// LS Electric XG5000 project: 8_22_1
// PLC LSPLC

PROGRAM NewProgram (task: 스캔 프로그램)

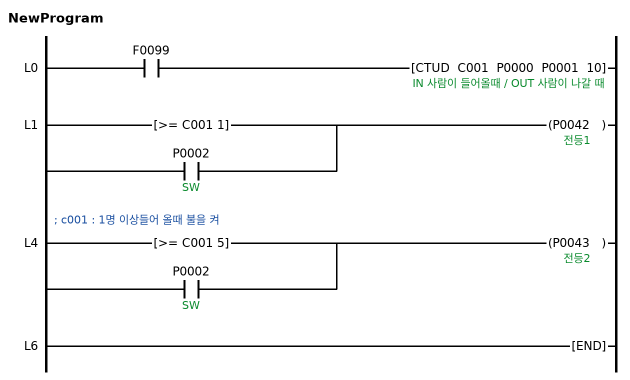
; L0
LOAD      F0099
CTUD      C001 P0000 P0001 10	// IN 사람이 들어올때 / OUT 사람이 나갈 때
; L1
LOAD>=    C001 1
OR        P0002	// SW
OUT       P0042	// 전등1
// c001 : 1명 이상들어 올때 불을 켜
; L4
LOAD>=    C001 5
OR        P0002	// SW
OUT       P0043	// 전등2
; L6
END